ABB RobotStudio station: ok.rsstn

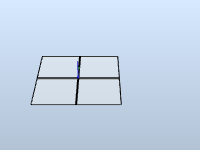
Station Station (saved by RobotStudio 6.5.7392.129)
Layout (positions relative to the parent item):
